// TIA Portal V20 export
ORGANIZATION_BLOCK "Main_1"   // OB1, LAD, ProgramCycle
TITLE = "Main Program Sweep (Cycle)"
{ S7_Optimized_Access := 'TRUE' }
// stored: SetENOAutomatically false
BEGIN

REGION Network 1
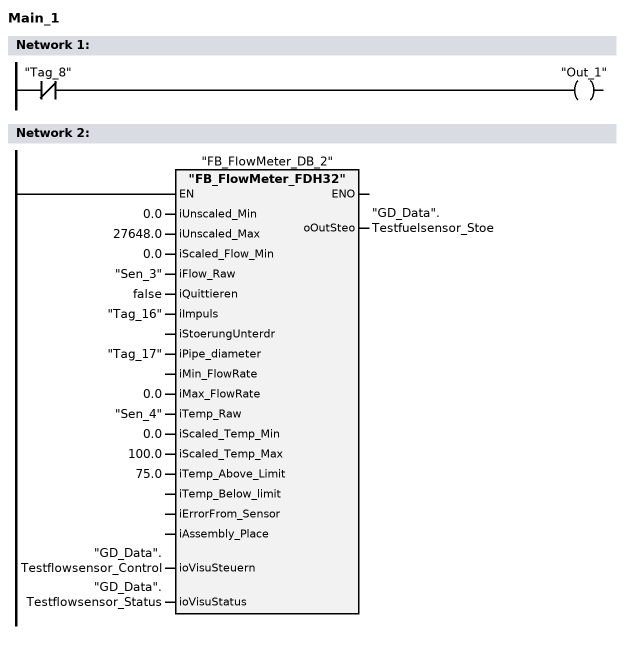
   RUNG wire#powerrail
      I_Contact( "Tag_8" )
      Coil( "Out_1" )
   END_RUNG
   // the same network as SCL:
   "Out_1" := NOT "Tag_8";
END_REGION

REGION Network 2
   RUNG wire#powerrail
      "FB_FlowMeter_DB_2"(iUnscaled_Min := 0.0, iUnscaled_Max := 27648.0, iScaled_Flow_Min := 0.0, iFlow_Raw := "Sen_3", iQuittieren := false, iImpuls := "Tag_16", iStoerungUnterdr :=, iPipe_diameter := "Tag_17", iMin_FlowRate :=, iMax_FlowRate := 0.0, iTemp_Raw := "Sen_4", iScaled_Temp_Min := 0.0, iScaled_Temp_Max := 100.0, iTemp_Above_Limit := 75.0, iTemp_Below_limit :=, iErrorFrom_Sensor :=, iAssembly_Place :=, ioVisuSteuern := "GD_Data".Testflowsensor_Control, ioVisuStatus := "GD_Data".Testflowsensor_Status, oOutSteo => "GD_Data".Testfuelsensor_Stoe)
   END_RUNG
   // the same network as SCL:
   "FB_FlowMeter_DB_2"(iUnscaled_Min := 0.0,   // "FB_FlowMeter_FDH32"
                       iUnscaled_Max := 27648.0,
                       iScaled_Flow_Min := 0.0,
                       iFlow_Raw := "Sen_3",
                       iQuittieren := false,
                       iImpuls := "Tag_16",
                       iPipe_diameter := "Tag_17",
                       iMax_FlowRate := 0.0,
                       iTemp_Raw := "Sen_4",
                       iScaled_Temp_Min := 0.0,
                       iScaled_Temp_Max := 100.0,
                       iTemp_Above_Limit := 75.0,
                       ioVisuSteuern := "GD_Data".Testflowsensor_Control,
                       ioVisuStatus := "GD_Data".Testflowsensor_Status,
                       oOutSteo => "GD_Data".Testfuelsensor_Stoe);
END_REGION
END_ORGANIZATION_BLOCK
